{attribute addProperty BoxType "AX8206-0000-0041-0041"}
{attribute addProperty Id "DeviceDevice_FD48B4B01620Ch_ACh_A_99F8614F240300Ch_BCh_B_5DC205AF240300WcStateAT %I*WcState_98A4DF7520.250InfoDataAT %I*InfoData_17277C5A208260"}
{attribute addProperty CRC "1253737747"}
{attribute addProperty SizeInBites "706"}
{attribute addProperty SizeInBytes "88.25"}
TYPE AX8206_C98B9CD1 :
STRUCT
	{attribute addProperty Name "Device"}
	Device : Device_FD48B4B0;
	{attribute addProperty Name "Ch_A"}
	Ch_A : Ch_A_99F8614F;
	{attribute addProperty Name "Ch_B"}
	Ch_B : Ch_B_5DC205AF;
	{attribute addProperty Name "WcState"}
	WcState : WcState_98A4DF75;
	{attribute addProperty Name "InfoData"}
	InfoData : InfoData_17277C5A;
END_STRUCT
END_TYPE

(* stored: Version 1.2.0.0, ProductVersion 3.1.4024.9
   DUT AX8206_C98B9CD1: Id {b8aadadb-eedb-4917-81c0-5e68958f749f} *)
